PROGRAM MAIN
VAR
END_VAR

END_PROGRAM

(* stored: Version 1.1.0.1
   POU MAIN: Id {1e048777-47af-4e33-bd66-1e639cad0451} *)
